(* PLC project Sin nombre, Desconocido Sin nombre 1 *)
(* stored: creationDateTime 2024-10-28T23:47:34, modificationDateTime 2024-10-29T13:08:26 *)

PROGRAM program0
  VAR
    sensor AT %IW0 : UINT;
  END_VAR
  VAR
    tope_normal : UINT := 34500;
    tope_alto : UINT := 36800;
    tope_superior : UINT := 38400;
    minimo_alto : UINT := 34501;
    minimo_superior : UINT := 36801;
    acumulador : UDINT := 38000;
  END_VAR
  VAR CONSTANT
    acumulador_prueba : UDINT := 35000;
    acumulador_prueba2 : UDINT := 36900;
  END_VAR
  VAR
    timer : BOOL := 1;
    verificar : BOOL := 0;
    timer_corrido : BOOL := 0;
    probar : BOOL := 0;
    acumular : BOOL := 0;
    entro : BOOL := 0;
    luz1 : BOOL := 0;  (* dar ubicacion *)
    luz2 : BOOL := 0;  (* dar ubicacion *)
    TP0 : TP;
    TOF1 : TOF;
    TP3 : TP;
    CTU_LINT0 : CTU_LINT;
    TP1 : TP;
    TOF0 : TOF;
    TOF2 : TOF;
  END_VAR
  VAR  (* added by the conversion: wires and edge detectors of the diagram *)
    _UINT_TO_UDINT81_ENO : BOOL;
    _UINT_TO_UDINT81_OUT : UDINT;
    _ADD78_ENO : BOOL;
    _ADD78_OUT : UDINT;
    R_TRIG1 : R_TRIG;
    _DIV87_OUT : ANY;
    _DIV87_ENO : BOOL;
    _UINT_TO_UDINT8_ENO : BOOL;
    _UINT_TO_UDINT8_OUT : UDINT;
    _GE93_ENO : BOOL;
    _GE93_OUT : BOOL;
    _UINT_TO_UDINT9_ENO : BOOL;
    _UINT_TO_UDINT9_OUT : UDINT;
    _LT100_ENO : BOOL;
    _LT100_OUT : BOOL;
    _UINT_TO_UDINT12_ENO : BOOL;
    _UINT_TO_UDINT12_OUT : UDINT;
    _GE104_ENO : BOOL;
    _GE104_OUT : BOOL;
    _AND127_ENO : BOOL;
    _AND127_OUT : BOOL;
    _OR129_ENO : BOOL;
    _OR129_OUT : BOOL;
  END_VAR

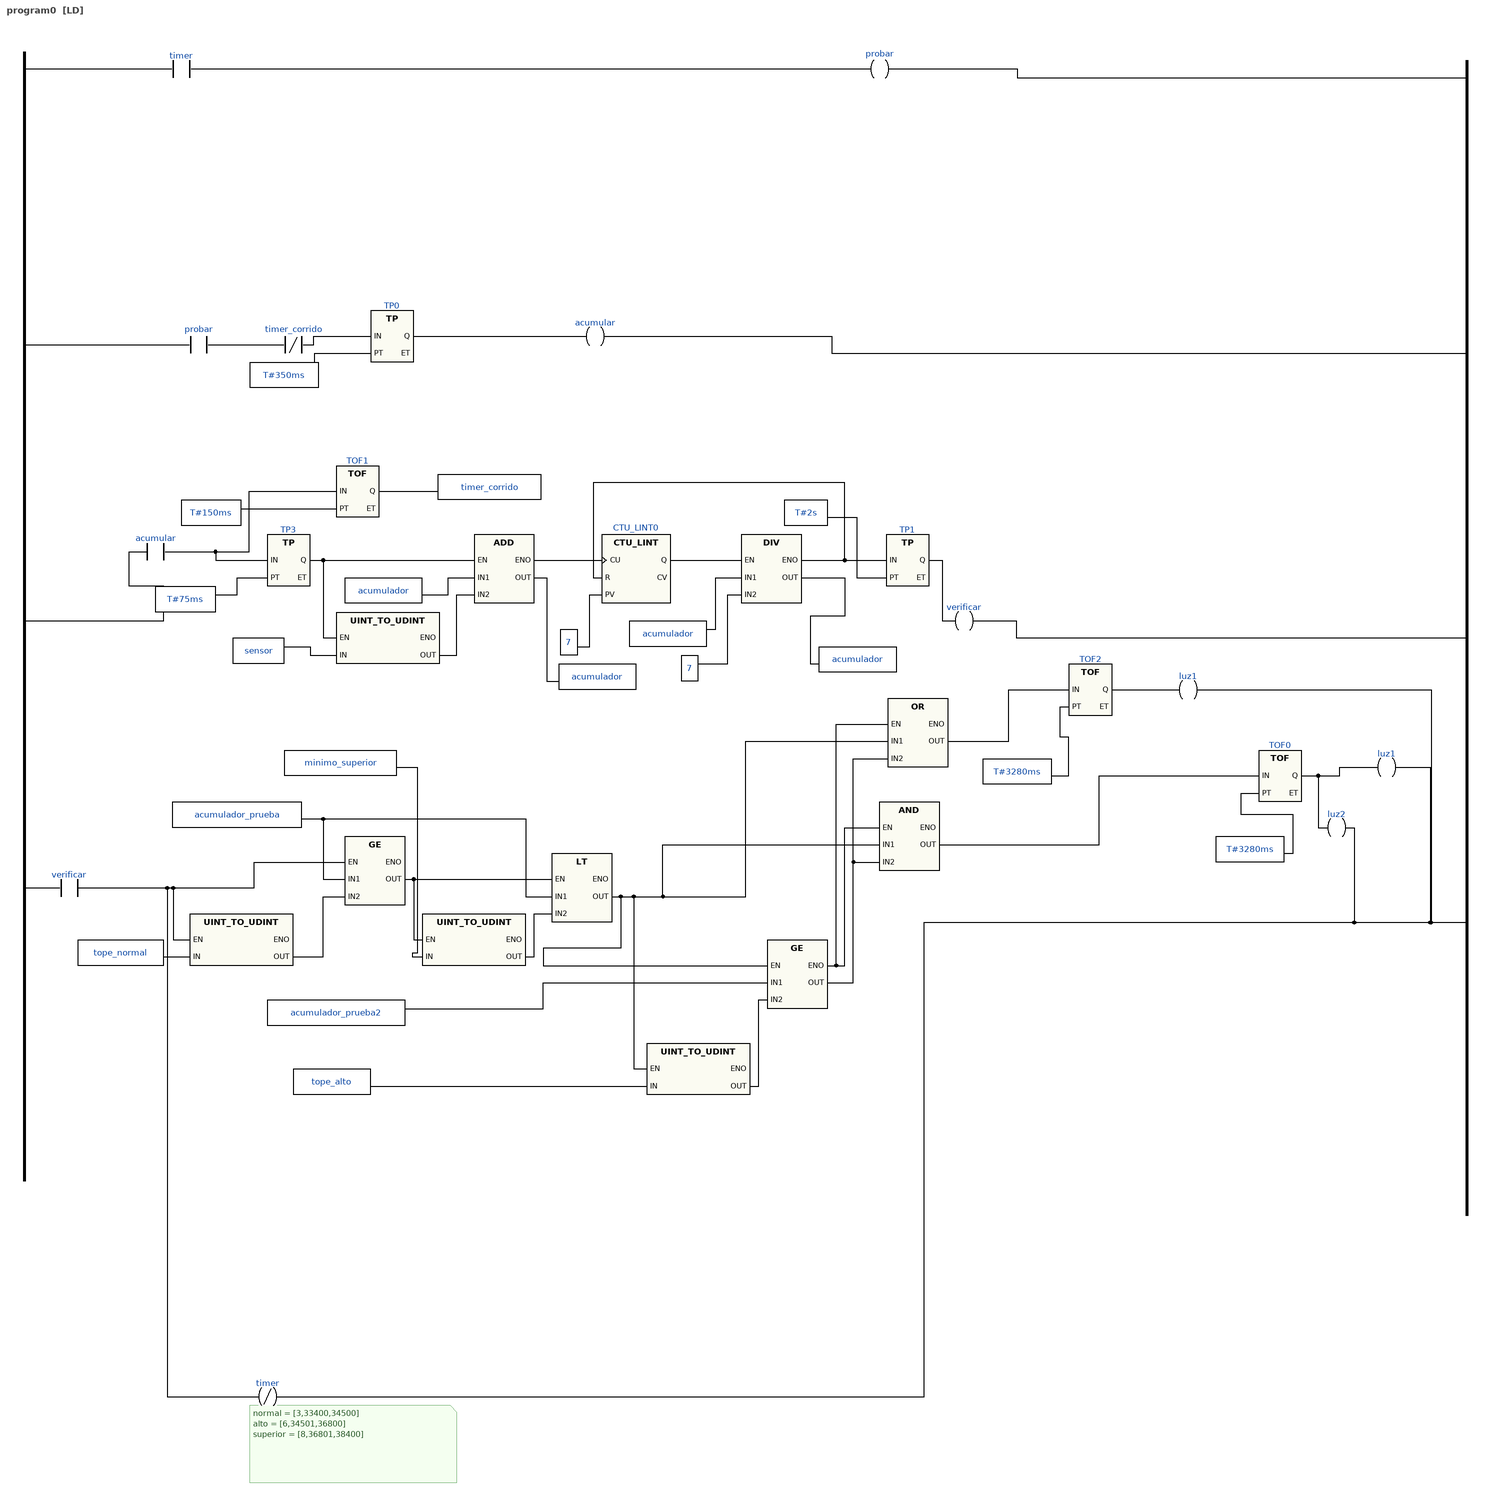
(* LD diagram, written out as Structured Text *)
probar := timer;
TP0(IN := probar AND NOT timer_corrido, PT := T#350ms);
acumular := TP0.Q;
TOF1(IN := acumular, PT := T#150ms);
timer_corrido := TOF1.Q;
TP3(IN := acumular, PT := T#75ms);
_UINT_TO_UDINT81_OUT := UINT_TO_UDINT(EN := TP3.Q, IN := sensor, ENO => _UINT_TO_UDINT81_ENO);
_ADD78_OUT := ADD(EN := TP3.Q, IN1 := acumulador, IN2 := _UINT_TO_UDINT81_OUT, ENO => _ADD78_ENO);
IF _ADD78_ENO THEN acumulador := _ADD78_OUT; END_IF;
R_TRIG1(CLK := _ADD78_ENO);
CTU_LINT0(CU := R_TRIG1.Q, R := _DIV87_OUT, PV := 7);
_DIV87_OUT := DIV(EN := CTU_LINT0.Q, IN1 := acumulador, IN2 := 7, ENO => _DIV87_ENO);
IF _DIV87_ENO THEN acumulador := _DIV87_OUT; END_IF;
timer := NOT verificar;
TP1(IN := _DIV87_ENO, PT := T#2s);
verificar := TP1.Q;
_UINT_TO_UDINT8_OUT := UINT_TO_UDINT(EN := verificar, IN := tope_normal, ENO => _UINT_TO_UDINT8_ENO);
_GE93_OUT := GE(EN := verificar, IN1 := acumulador_prueba, IN2 := _UINT_TO_UDINT8_OUT, ENO => _GE93_ENO);
_UINT_TO_UDINT9_OUT := UINT_TO_UDINT(EN := _GE93_OUT, IN := minimo_superior, ENO => _UINT_TO_UDINT9_ENO);
_LT100_OUT := LT(EN := _GE93_OUT, IN1 := acumulador_prueba, IN2 := _UINT_TO_UDINT9_OUT, ENO => _LT100_ENO);
_UINT_TO_UDINT12_OUT := UINT_TO_UDINT(EN := _LT100_OUT, IN := tope_alto, ENO => _UINT_TO_UDINT12_ENO);
_GE104_OUT := GE(EN := _LT100_OUT, IN1 := acumulador_prueba2, IN2 := _UINT_TO_UDINT12_OUT, ENO => _GE104_ENO);
_AND127_OUT := AND(EN := _GE104_ENO, IN1 := _LT100_OUT, IN2 := _GE104_OUT, ENO => _AND127_ENO);
TOF0(IN := _AND127_OUT, PT := T#3280ms);
luz2 := TOF0.Q;
luz1 := TOF0.Q;
_OR129_OUT := OR(EN := _GE104_ENO, IN1 := _LT100_OUT, IN2 := _GE104_OUT, ENO => _OR129_ENO);
TOF2(IN := _OR129_OUT, PT := T#3280ms);
luz1 := TOF2.Q;
(* normal = [3,33400,34500] 
alto = [6,34501,36800]
superior = [8,36801,38400] *)
END_PROGRAM

CONFIGURATION Config0
  RESOURCE Res0 ON PLC
    TASK task0(INTERVAL := T#20ms, PRIORITY := 0);
    PROGRAM instance0 WITH task0 : program0;
  END_RESOURCE
END_CONFIGURATION
